PROGRAM MAIN
VAR
END_VAR

END_PROGRAM

(* stored: Version 1.1.0.1
   POU MAIN: Id {6db1c2aa-9afd-444d-bbb2-ac8aed5fb808} *)
